// TIA Portal V16 export
// export: Created 2021-11-12T13:32:40.0102614Z, ExportSetting WithDefaults, DisplayName Totally Integrated Automation Portal, DisplayVersion V16 Update 3, DisplayName TIA Portal Version Control Interface, DisplayVersion V16 Update 2, DisplayName TIA Portal Openness, DisplayVersion V16 Update 3, DisplayName SINAMICS Startdrive Advanced, DisplayVersion V16 Update 5, DisplayName SINAMICS Startdrive G130, G150, S120, S150, SINAMICS MV, S210, DisplayVersion V16 Update 5, DisplayName SINAMICS Startdrive G110M, G120, G120C, G120D, G120P, G115D, DisplayVersion V16 Update 5, DisplayName STEP 7 Professional, DisplayVersion V16 Update 3, DisplayName STEP 7 Safety, DisplayVersion V16, DisplayName WinCC UA Professional, DisplayVersion V16 Update 3
DATA_BLOCK "STATUS_2R2"   // DB2115
{ S7_Optimized_Access := 'TRUE' }
VERSION : 0.1
// stored: AutoNumber false, DBAccessibleFromOPCUA true, IsOnlyStoredInLoadMemory false, IsRetainMemResEnabled false, IsWriteProtectedInAS false, MemoryReserve 100
   VAR
      xxxxx___BinarySensors___xxxxx : Byte;
      "CM01-BL01_4" : Bool;   // Proplachovací nádrž 2 Vysoká hladina Varování
      "CM01-BL01_5" : Bool;   // Proplachovací nádrž 2 Vysoká hladina Max
      xxxxx___BinaryOthers___xxxxx : Byte;
      PwrOK : Bool;
      "000UH11-SF13" : Bool;   // Okamžitý stop Robot 2R2
      "000UH11-SF10" : Bool;   // Robot 2R2 Proplach
      "000UH11-SF11" : Bool;   // Robot 2R2 Nástřik
      xxxxx___AnalogueSensors___xxxxx : Byte;
      xxxxx___Drives___xxxxx : Byte;
      RO01 : Struct   // Robot
         Main : "UDT_Status_main";
         Specific : "UDT_RobotABB_Status_specific";
         Error : "UDT_Error01";
      END_STRUCT;
      RC01 : Struct   // Controller
         Main : "UDT_Status_main";
         Specific : "UDT_DriveRobotABB_Status_specific";
         Error : "UDT_Error01";
      END_STRUCT;
      Lubricating : Struct   // Lubricating
         Main : "UDT_Status_main";
         Specific : "UDT_DriveRobotABB_Status_specific";
         Error : "UDT_Error01";
      END_STRUCT;
      xxxxx___Others___xxxxx : Byte;
      Interlocks : "UDT_RobotABB_Interlock";
      ZoneRelease : "UDT_RobotABB_ZoneReleaseToRobot";
      xxxxx___Alarms___xxxxx : Byte;
      RO01_Timeout : Struct   // Robot job active for too long / Job robota aktivní příliš dlhou dobu.
         Main { S7_SetPoint := 'True'} : "UDT_Status_main";
         Specific { S7_SetPoint := 'True'} : "UDT_DI_Mon_Status_specific";
         Error { S7_SetPoint := 'True'} : "UDT_Error01";
      END_STRUCT;
      RO01_LubStartErr : Struct   // Lubrication job did not start (robot did not move)
         Main { S7_SetPoint := 'True'} : "UDT_Status_main";
         Specific { S7_SetPoint := 'True'} : "UDT_DI_Mon_Status_specific";
         Error { S7_SetPoint := 'True'} : "UDT_Error01";
      END_STRUCT;
      "CM01-BL01_4_alarm" : Struct   // Flush tank 2 - high level error. / Proplachovací nádrž 2 Vysoká hladina Varování
         Main : "UDT_Status_main";
         Specific : "UDT_DI_Mon_Status_specific";
         Error : "UDT_Error01";
      END_STRUCT;
      "CM01-BL01_5_alarm" : Struct   // Flush tank 2 - high level warning. / Proplachovací nádrž 2 Vysoká hladina Max
         Main : "UDT_Status_main";
         Specific { S7_SetPoint := 'True'} : "UDT_DI_Mon_Status_specific";
         Error { S7_SetPoint := 'True'} : "UDT_Error01";
      END_STRUCT;
      xxxxx___SftyAlarms___xxxxx_1 : Byte;
      ES : Struct   // E-stop
         Main { S7_SetPoint := 'True'} : "UDT_Status_main";
         Specific { S7_SetPoint := 'True'} : "UDT_DI_Mon_Status_specific";
         Error { S7_SetPoint := 'True'} : "UDT_Error01";
      END_STRUCT;
   END_VAR
BEGIN
END_DATA_BLOCK
